// TIA Portal V17 export
// export: Created 2024-08-20T13:26:11.2767376Z, ExportSetting WithDefaults, DisplayName Totally Integrated Automation Portal, DisplayVersion V17 Update 4, DisplayName TIA Portal Openness, DisplayVersion V17 Update 4, DisplayName TIA Portal Version Control Interface, DisplayVersion V17, DisplayName STEP 7 Professional, DisplayVersion V17 Update 4, DisplayName STEP 7 Safety, DisplayVersion V17, DisplayName WinCC Advanced, DisplayVersion V17 Update 4
DATA_BLOCK "PDIR_DB_MB-01"   // DB422
VERSION : 0.1
// stored: AutoNumber false, DBAccessibleFromOPCUA true, InstanceOfName PDIR, InstanceOfType FB
"PDIR"
   // VAR_INPUT
   //    ML : Bool;
   //    MR : Bool;
   //    DL : Bool;
   //    MF1 : Bool;
   //    MF2 : Bool;
   //    HM : Bool;
   //    HA : Bool;
   //    CMA : Bool;
   //    CLM : Bool;
   //    CDM : Bool;
   //    CRF : Bool;
   //    CRTO : Bool;
   //    CL1S : Bool;
   // END_VAR
   // VAR_OUTPUT
   //    YFPP : Bool;
   //    YF : Bool;
   //    CL : Bool;
   // END_VAR
   // VAR_IN_OUT
   //    SEG : Int;
   //    MIN : Int;
   //    HOR : Int;
   // END_VAR
   // VAR
   //    AUX01 : Bool;
   //    AUX02 : Bool;
   //    AUX03 : Bool;
   //    AUX04 : Bool;
   //    AUX05 : Bool;
   //    AUX06 : Bool;
   //    AUX07 : Bool;
   //    AUX08 : Bool;
   //    AUX09 : Bool;
   //    P60S : Bool;
   //    P60M : Bool;
   //    PFHO : Bool;
   //    TPP1 { S7_SetPoint := 'True'} : TON_TIME;
   //    TPP2 { S7_SetPoint := 'True'} : TON_TIME;
   // END_VAR
BEGIN
END_DATA_BLOCK
